{attribute 'qualified_only'}
{attribute 'strict'}
TYPE BEAMLINE :
(
    None := 0,
    Soft := 1,
    Hard := 2
) UINT;
END_TYPE

(* stored: Version 1.1.0.1
   DUT BEAMLINE: Id {b306946f-4b63-4652-812b-42c4fb2c08cb} *)
